// TIA Portal project "databloklarlatankvana" (V20)

(* hardware
DEVICE "S7-1200 station_1"  S7-1200 Station
   slot 0: "Rack_0"  S7-1200 Rack  Rack  V1.0
   slot 1: "PLC_1"  CPU 1214C DC/DC/Rly  6ES7 214-1HG40-0XB0  V4.7
*)

// ===== PLC "PLC_1"  CPU 1214C DC/DC/Rly =====

VAR_GLOBAL   // PLC tag table "Default tag table"
   "start but 1" AT %I0.0 : Bool;
   "stop but 1" AT %I0.1 : Bool;
   "üst sensör 1" AT %I0.2 : Bool;
   "alt sensör 1" AT %I0.3 : Bool;
   "vana 1" AT %Q0.0 : Bool;
   "start but 2" AT %I0.4 : Bool;
   "stop but 2" AT %I0.5 : Bool;
   "üst sensör 2" AT %I0.6 : Bool;
   "alt sensör 2" AT %I0.7 : Bool;
   "vana 2" AT %Q0.1 : Bool;
END_VAR

DATA_BLOCK "doldurma vanası 1"   // DB1
{ S7_Optimized_Access := 'TRUE' }
VERSION : 0.1
// stored: InstanceOfName doldurma vanası
"doldurma vanası"
BEGIN
END_DATA_BLOCK

DATA_BLOCK "doldurma vanası 2"   // DB2
{ S7_Optimized_Access := 'TRUE' }
VERSION : 0.1
// stored: InstanceOfName doldurma vanası
"doldurma vanası"
BEGIN
END_DATA_BLOCK

FUNCTION_BLOCK "doldurma vanası"   // FB1, LAD
{ S7_Optimized_Access := 'TRUE' }
VERSION : 0.1
   VAR_INPUT
      start : Bool;
      stop : Bool;
      "üst seviye" : Bool;
      "alt seviye" : Bool;
   END_VAR
   VAR_OUTPUT
      "vana çalıştır" : Bool;
   END_VAR
   VAR
      "vana merker 1" : Bool;
      "vana merker 2" : Bool;
   END_VAR
BEGIN

REGION Network 1
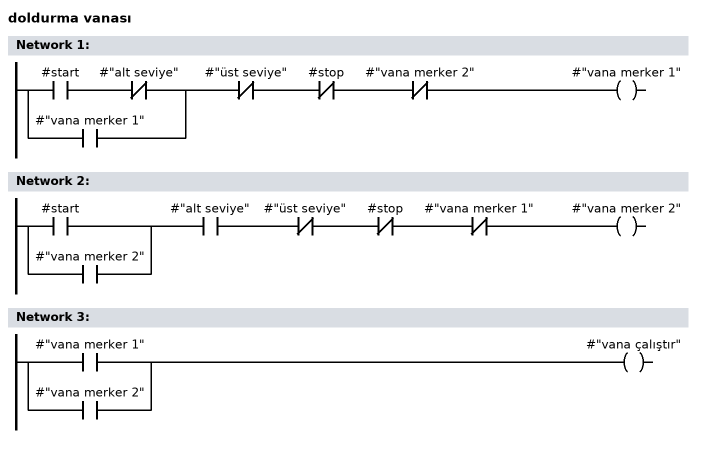
   RUNG wire#powerrail
      Contact( #start )
      I_Contact( #"alt seviye" )
      wire#w1
      I_Contact( #"üst seviye" )
      I_Contact( #stop )
      I_Contact( #"vana merker 2" )
      Coil( #"vana merker 1" )
   END_RUNG
   RUNG wire#powerrail
      Contact( #"vana merker 1" )
   END_RUNG wire#w1
   // the same network as SCL:
   #"vana merker 1" := ((#start AND NOT #"alt seviye") OR #"vana merker 1") AND NOT #"üst seviye" AND NOT #stop AND NOT #"vana merker 2";
END_REGION

REGION Network 2
   RUNG wire#powerrail
      Contact( #start )
      wire#w1
      Contact( #"alt seviye" )
      I_Contact( #"üst seviye" )
      I_Contact( #stop )
      I_Contact( #"vana merker 1" )
      Coil( #"vana merker 2" )
   END_RUNG
   RUNG wire#powerrail
      Contact( #"vana merker 2" )
   END_RUNG wire#w1
   // the same network as SCL:
   #"vana merker 2" := (#start OR #"vana merker 2") AND #"alt seviye" AND NOT #"üst seviye" AND NOT #stop AND NOT #"vana merker 1";
END_REGION

REGION Network 3
   RUNG wire#powerrail
      Contact( #"vana merker 1" )
      wire#w1
      Coil( #"vana çalıştır" )
   END_RUNG
   RUNG wire#powerrail
      Contact( #"vana merker 2" )
   END_RUNG wire#w1
   // the same network as SCL:
   #"vana çalıştır" := #"vana merker 1" OR #"vana merker 2";
END_REGION
END_FUNCTION_BLOCK

ORGANIZATION_BLOCK "Main"   // OB1, LAD, ProgramCycle
TITLE = "Main Program Sweep (Cycle)"
{ S7_Optimized_Access := 'TRUE' }
VERSION : 0.1
   VAR_INPUT
      Initial_Call : Bool;   // Initial call of this OB
      Remanence : Bool;   // =True, if remanent data are available
   END_VAR
BEGIN

REGION Network 1
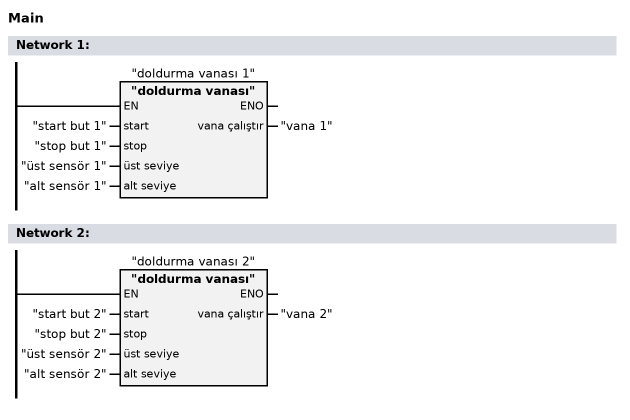
   RUNG wire#powerrail
      "doldurma vanası 1"(start := "start but 1", stop := "stop but 1", "üst seviye" := "üst sensör 1", "alt seviye" := "alt sensör 1", "vana çalıştır" => "vana 1")
   END_RUNG
   // the same network as SCL:
   "doldurma vanası 1"(start := "start but 1",   // "doldurma vanası"
                       stop := "stop but 1",
                       "üst seviye" := "üst sensör 1",
                       "alt seviye" := "alt sensör 1",
                       "vana çalıştır" => "vana 1");
END_REGION

REGION Network 2
   RUNG wire#powerrail
      "doldurma vanası 2"(start := "start but 2", stop := "stop but 2", "üst seviye" := "üst sensör 2", "alt seviye" := "alt sensör 2", "vana çalıştır" => "vana 2")
   END_RUNG
   // the same network as SCL:
   "doldurma vanası 2"(start := "start but 2",   // "doldurma vanası"
                       stop := "stop but 2",
                       "üst seviye" := "üst sensör 2",
                       "alt seviye" := "alt sensör 2",
                       "vana çalıştır" => "vana 2");
END_REGION
END_ORGANIZATION_BLOCK